FUNCTION projArray1: ARRAY[0..4] of DINT
VAR_INPUT
    arr: ARRAY[0..1] of ARRAY[0..4] of DINT;
    idx: DINT;
END_VAR


        projArray1 := arr[normProjIdx(idx, 2)];

END_FUNCTION

(* stored: ProductVersion 3.1.0.18, Version 1.1.0.1 *)
